FUNCTION_BLOCK SomeCyclicClass
VAR
	_myWriter : ITF_Writer;
END_VAR

METHOD DoSomething : BOOL
VAR_INPUT
END_VAR
///////Perform some operations////////

IF _myWriter <> 0 THEN
	_myWriter.WriteMessage('I did a job :-)');
END_IF
END_METHOD

PROPERTY MyWriter : ITF_Writer
GET
MyWriter := _myWriter;
END_GET
SET
_myWriter := MyWriter;
END_SET
END_PROPERTY

END_FUNCTION_BLOCK

(* stored: Version 1.1.0.1, ProductVersion 3.1.4024.12
   POU SomeCyclicClass: Id {c971e421-8128-48df-a9ae-39d00c83f57b}, SpecialFunc None
   Method DoSomething: Id {565c603a-7b40-431c-b568-38c5684d96f6}
   Property MyWriter: Id {7ad904d8-f5a6-4abc-8725-2587f58609e4}
   Get Get: Id {51d8146f-cd4a-4e35-9bf6-60a75ad22deb}
   Set Set: Id {af74eea1-a8e5-4e91-96bb-88c67c2c27c9} *)
